TYPE ST_CmdContent :
STRUCT
	SysTime				: STRING;
	Source				: STRING;
	Command				: STRING;
END_STRUCT
END_TYPE

(* stored: Version 1.1.0.1, ProductVersion 3.1.4024.13
   DUT ST_CmdContent: Id {c6bc7f34-5020-44c7-acb4-834e299ada40} *)
